{attribute addProperty BoxType "KL2732"}
{attribute addProperty Id "Channel_1Channel_E75BD82E00Channel_2Channel_E75BD82E00"}
{attribute addProperty CRC "1288439370"}
{attribute addProperty SizeInBites "0"}
{attribute addProperty SizeInBytes "0"}
TYPE KL2732_4CCC064A :
STRUCT
	{attribute addProperty Name "Channel_1"}
	Channel_1 : Channel_E75BD82E;
	{attribute addProperty Name "Channel_2"}
	Channel_2 : Channel_E75BD82E;
END_STRUCT
END_TYPE

(* stored: Version 1.2.0.0, ProductVersion 3.1.4024.9
   DUT KL2732_4CCC064A: Id {4973a6f2-e2f7-4e20-9b67-c6ab58b60b26} *)
